FUNCTION_BLOCK FB_HMI_METIS_RH_SENSOR EXTENDS FB_HMI_COMPONENT
VAR_INPUT
END_VAR
VAR_OUTPUT
END_VAR
VAR_IN_OUT
    fbInstance : FB_METIS_RH_SENSOR;
END_VAR
VAR
END_VAR

fbHealthStatus(
    bIsEnabled := fbInstance.stat.bValid,
    bIsGood := NOT fbInstance.stat.bError);

fbBusyStatus(
    bIsEnabled := FALSE,
    bIsBusy := FALSE);

M_UpdateStatusColor();

END_FUNCTION_BLOCK

(* stored: Version 1.1.0.1, ProductVersion 3.1.4024.14
   POU FB_HMI_METIS_RH_SENSOR: Id {f041fcef-4fa1-4701-b271-c2beddccbd1e}, SpecialFunc None *)
